Staubli VAL3: OnF6.pgx

program OnF6()
  local num l_i
  local string l_sMsg
  local string l_sYesNo[2]
begin
  //重新载入数据，所有做过的修改都不保存
  l_sYesNo[0]="是"
  l_sYesNo[1]="否"
  l_sMsg="重载会删除所有修改，请确认!"
  call user:questionDialog(l_sMsg,l_sYesNo,l_i)
  if l_i==0 or l_i==1
    call JTP()
    popUpMsg("重载数据完成")
    logMsg("重载数据完成")
  endIf
  bUserRefresh=true
end
